FUNCTION ARR08B_TO_WORDS_BE (* this Function extracts the 4 WORD from a 8-BYTE Array *)
  (* Standard: 61499-1; Description: Copyright (c) 2024 HR Agrartechnik GmbH This program and the accompanying materials are made available under the terms of the Eclipse Public License 2.0 which is available at https://www.eclipse.org/legal/epl-2.0/ SPDX-License-Identifier: EPL-2.0 *)
  (* Version 1.0, 2024-02-22, Franz Höpfinger, HR Agrartechnik GmbH *)
  PACKAGE logiBUS::utils::conversion::arr::forwarding;
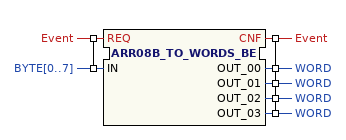
  EVENT_INPUT
    REQ WITH IN;
  END_EVENT
  EVENT_OUTPUT
    CNF WITH OUT_00, OUT_01, OUT_02, OUT_03;
  END_EVENT
  VAR_INPUT
    IN : ARRAY [0..7] OF BYTE; (* ARR08B Input *)
  END_VAR
  VAR_OUTPUT
    OUT_00 : WORD; (* WORD 00 *)
    OUT_01 : WORD; (* WORD 01 *)
    OUT_02 : WORD; (* WORD 02 *)
    OUT_03 : WORD; (* WORD 03 *)
  END_VAR
  BODY IN ST:
PACKAGE logiBUS::utils::conversion::arr::forwarding;

(* this Function extracts the 4 WORD from a 8-BYTE Array *)
FUNCTION ARR08B_TO_WORDS_BE

VAR_INPUT
	IN : ARRAY[0..7] OF BYTE; // ARR08B Input
END_VAR

VAR_OUTPUT
	OUT_00 : WORD; // WORD 00
	OUT_01 : WORD; // WORD 01
	OUT_02 : WORD; // WORD 02
	OUT_03 : WORD; // WORD 03
END_VAR

OUT_00.%B1 := IN[0];
OUT_00.%B0 := IN[1];
OUT_01.%B1 := IN[2];
OUT_01.%B0 := IN[3];
OUT_02.%B1 := IN[4];
OUT_02.%B0 := IN[5];
OUT_03.%B1 := IN[6];
OUT_03.%B0 := IN[7];

END_FUNCTION
  END_BODY
END_FUNCTION
